(* IEC 61131-3 sources: CodesysTest/export/Pro24.dev/Plc Logic/Application/Pro24/Applied Motion/FB_AppliedMotionStepServoEIPBase.pou, 2 files *)

(* ---- MoveToPositionTorque.m.st ---- *)
(*#-#-#-#-#-#-#-#-#-#---Declaration---#-#-#-#-#-#-#-#-#-#-#-#-#*)

METHOD MoveToPositionTorque
VAR_INPUT
	(*Position to move to in inches*)
    position    : REAL;
    (*Acceleration in RPM/sec*)
    acceleration    : INT;
    (*Deceleration in RPM/sec*)
    deceleration    : INT;
    (*Velocity in .25RPM*)
    velocity    : INT;
	(*Current in .01A*)
	current : DINT;
END_VAR
(*#-#-#-#-#-#-#-#-#-#---Implementation---#-#-#-#-#-#-#-#-#-#-#-#-#*)

commandSuccessful := FALSE;

distanceToMoveInSteps := REAL_TO_DINT((position) * stepsPerInchSetpoint);
IF reversePolarity THEN
    distanceToMoveInSteps := distanceToMoveInSteps * -1;
END_IF

pointToPointAccelSetpoint := acceleration;
pointToPointDecelSetpoint := deceleration;
velocitySetpoint := velocity;
currentLimit := current;

commands.feedToPosition := TRUE;

(* ---- ResetEncoderPosition.m.st ---- *)
(*#-#-#-#-#-#-#-#-#-#---Declaration---#-#-#-#-#-#-#-#-#-#-#-#-#*)

METHOD ResetEncoderPosition
VAR_INPUT
END_VAR
(*#-#-#-#-#-#-#-#-#-#---Implementation---#-#-#-#-#-#-#-#-#-#-#-#-#*)

THIS^.ExecuteStoredProgram(9);
